// TIA Portal V17 export
// export: Created 2026-05-13T16:54:41.7289132Z, ExportSetting WithDefaults, DisplayName Totally Integrated Automation Portal, DisplayVersion V17 Update 4, DisplayName TIA Portal Openness, DisplayVersion V17 Update 4, DisplayName TIA Portal Version Control Interface, DisplayVersion V17, DisplayName SINAMICS Startdrive Advanced, DisplayVersion V17, DisplayName SINAMICS Startdrive G130, G150, S120, S150, SINAMICS MV, S210, DisplayVersion V17, DisplayName SINAMICS Startdrive G110M, G120, G120C, G120D, G120P, G115D, DisplayVersion V17, DisplayName STEP 7 Professional, DisplayVersion V17 Update 4, DisplayName STEP 7 Safety, DisplayVersion V17, DisplayName WinCC Professional, DisplayVersion V17 Update 4
TagTable "CS"
  CS_MS模式设定 : Real  (PLC tag CS.MS模式设定, HMI_连接_1, 100 ms)
  CS_CM触摸屏运行启动 : Bool  (PLC tag CS.CM触摸屏运行启动, HMI_连接_1, 100 ms)
  CS_AQ安全停机 : Bool  (PLC tag CS.AQ安全停机, HMI_连接_1, 100 ms)
  CS_SD手动模式 : Bool  (PLC tag CS.SD手动模式, HMI_连接_1, 100 ms)
  CS_SF送风机动画 : Int  (PLC tag CS.SF送风机动画, HMI_连接_1, 100 ms)
  CS_YF引风机动画 : Int  (PLC tag CS.YF引风机动画, HMI_连接_1, 100 ms)
  CS_JL进料泵动画 : Int  (PLC tag CS.JL进料泵动画, HMI_连接_1, 100 ms)
  CS_JB搅拌电机动画 : Int  (PLC tag CS.JB搅拌电机动画, HMI_连接_1, 100 ms)
  CS_ZD自动模式 : Bool  (PLC tag CS.ZD自动模式, HMI_连接_1, 100 ms)
  CS_主管道动画 : Bool  (PLC tag CS.主管道动画, HMI_连接_1, 100 ms)
